FUNCTION_BLOCK Tank IMPLEMENTS I_Domain, I_Execute
VAR_INPUT
	bEnable			: BOOL;
	fLevel			: REAL;
END_VAR
VAR_OUTPUT
	bInletValveOpen		: BOOL;
END_VAR
VAR_STAT
	nId				: UDINT;
END_VAR
VAR CONSTANT
	MAX_STATE		: UDINT := 6;
END_VAR
VAR
	exe				: Execute(THIS^);

	// Context
	ctx				: Tank_Ctx;
	A_DomTag		: A_Tag(domTag, ctx.priv.iDomTag);
	
	// State Machine
	
	stateMachine	: StateMachine;
	stateRepo		: StateRepo<MAX_STATE>;
	stateBuffer		: StateBuffer<MAX_STATE>;
	stateMgr		: StateManager<MAX_STATE>(stateMachine, stateRepo, stateBuffer);
	A_Smgr			: A_StateManager(stateMgr, ctx.priv.smgr);
	
	// States
	
	Disabled			: Tank_Disabled(stateRepo, ctx);
	A_Disabled			: A_Tag(Disabled.Tag, ctx.state.iDisabled);
	
	Enabled				: Tank_Enabled(stateRepo, ctx);
	A_Enabled			: A_Tag(Enabled.Tag, ctx.state.iEnabled);
	
	Fault				: Tank_Fault(stateRepo, ctx);
	A_Fault				: A_Tag(Fault.Tag, ctx.state.iFault);
	
	Fill				: Tank_Fill(stateRepo, ctx);
	A_Fill				: A_Tag(Fill.Tag, ctx.state.iFill);
	
	SystemOff			: Tank_SystemOff(stateRepo, ctx);
	A_SystemOff			: A_Tag(SystemOff.Tag, ctx.state.iSystemOff);
	
	// FLAGS
	flagList		: FlagList<2>;
	A_IsFillable	: A_Flag(flagList, ctx.priv.IsFillable);
	A_IsEmpty		: A_Flag(flagList, ctx.priv.IsEmpty);
	
	// SIGNALS
	signalList		: SignalList<0>;
	A_SmgrChange	: A_Signal(signalList, stateMgr.GetOnChange());
	A_Request		: A_Signal(signalList, ctx.priv.Request);
	
	// RECEIVERS
	receiverList	: ReceiverList<0>;
	
	// HMI
	statusText		: Tank_StatusText(ctx);
	
	// DOMAIN
	domTag			: Tag;
	domain			: Domain(domTag, stateMgr, flagList, signalList, receiverList);
	
	// PRIV
	bInit			: BOOL := TRUE;
END_VAR

METHOD Execute
IF bInit THEN
	IF IsErr(FindFlag(ctx.priv.iTankCtrl.Flags, 'IsSystemOn', iFlag => ctx.priv.iIsSystemOn)) THEN
		DebugMsg(THIS^, 'Missing iIsSystemOn!');
	END_IF
	
	IF IsErr(FindRec(ctx.priv.iTankCtrl.Recs, 'OnRequest', iRec => ctx.priv.iRequestReceiver)) THEN
		DebugMsg(THIS^, 'Missing iRequestReceiver!');
	END_IF

	ctx.priv.smgr.Request(ctx.state.iDisabled);	

	bInit := FALSE;
END_IF

IF fLevel <= ctx.hmi.fLowLevel.val THEN
	ctx.priv.IsEmpty.Rise();
ELSE
	ctx.priv.IsEmpty.Lower();
END_IF

// INPUTS
ctx.io.in.bEnable := bEnable;
ctx.io.in.fLevel := fLevel;

// OUTPUTS
bInletValveOpen := ctx.io.out.bInletValveOpen;
END_METHOD

//FB_Init is always available implicitly and it is used primarily for initialization.
//The return value is not evaluated. For a specific influence, you can also declare the
//methods explicitly and provide additional code there with the standard initialization
//code. You can evaluate the return value.
METHOD FB_Init: BOOL
VAR_INPUT
    bInitRetains: BOOL; // TRUE: the retain variables are initialized (reset warm / reset cold)
    bInCopyCode: BOOL;  // TRUE: the instance will be copied to the copy code afterward (online change)
	
	iTankCtrlDom		: I_Domain;
END_VAR
domTag.Option := UDINT_TO_STRING((nId := nId + 1));
ctx.priv.iTankCtrl := iTankCtrlDom;
END_METHOD

PROPERTY Flags : Domains.Flags.I_FlagList
GET
Flags := flagList;
END_GET
END_PROPERTY

PROPERTY Recs : Domains.Broadcast.I_ReceiverList
GET
Recs := receiverList;
END_GET
END_PROPERTY

PROPERTY Signals : Domains.Broadcast.I_SignalList
GET
Signals := signalList;
END_GET
END_PROPERTY

PROPERTY Smgr : Domains.States.I_StateManager
GET
Smgr := stateMgr;
END_GET
END_PROPERTY

PROPERTY Tag : Tags.I_Tag
GET
Tag := domTag;
END_GET
END_PROPERTY

METHOD ToDebug : Debug.I_Debug
ToDebug := THIS^;
END_METHOD

END_FUNCTION_BLOCK

(* stored: Version 1.1.0.1
   POU Tank: Id {a786dec2-6939-4565-9772-0b044609bff7}, SpecialFunc None
   Method Execute: Id {ef7225f4-9ca0-4312-9418-cb00cb75b449}
   Method FB_init: Id {26ecba72-b5e5-47a7-8e25-327ca4a99a62}
   Property Flags: Id {b797542f-79c7-4f97-90ef-c0e4ad10e674}
   Get Get: Id {11a6da6c-09f9-4bea-8a0f-4f011805818e}
   Property Recs: Id {2c46d922-634c-4b5d-ad13-9652dd6b287c}
   Get Get: Id {14c8e575-5afd-4a3d-b739-802d2f5c791e}
   Property Signals: Id {2b6c7e42-0fef-4fc3-87e7-d7e1d8a92c82}
   Get Get: Id {c41b3a2c-b918-452b-93f2-0e88f812ebc4}
   Property Smgr: Id {2ba05b8c-beba-4d32-b7c8-11d3af92314f}
   Get Get: Id {0a2a2d58-c216-4c58-af7e-f1cb066c32b7}
   Property Tag: Id {98ac75f8-e8ad-4fd8-8513-ffa86bdcf2fa}
   Get Get: Id {591d43d6-3408-4f73-8768-ab4de5af6ff3}
   Method ToDebug: Id {9c1b2447-c187-4a9e-adf9-f9f8c006ebf6} *)
